FUNCTION_BLOCK SawMotor (* goFB_ignore *)
  (* Standard: 61499-2 *)
  (* Version 0.1, 2017-00-16, hpea485, UOA *)
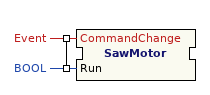
  EVENT_INPUT
    CommandChange WITH Run;
  END_EVENT
  VAR_INPUT
    Run : BOOL;
  END_VAR
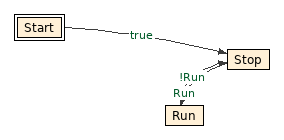
  EC_STATES
    Start;
    Run;
    Stop;
  END_STATES
  EC_TRANSITIONS
    Start TO Stop := true;
    Run TO Stop := !Run;
    Stop TO Run := Run;
  END_TRANSITIONS
END_FUNCTION_BLOCK
